FUNCTION_BLOCK FB_IFM_PN2x99
VAR_INPUT
	Grenzwert:REAL; //Grenzwer für HMI Blinken
END_VAR
VAR_OUTPUT
END_VAR
VAR
	IOData AT %I*:INT;
	V12 AT %Q*:BOOL;
	V14 AT %Q*:BOOL;
	
	IOData2:INT;
	Druck:REAL; //mbar (-1000 to 1100)
	OUT1:BOOL;
	OUT2:BOOL;
	
	state:INT:=1;
END_VAR

OUT1:=GETBIT32(inVal32:= IOData, bitNo:= 0);
OUT2:=GETBIT32(inVal32:= IOData, bitNo:= 1);

IOData2:=(IOData/4);
Druck:=INT_TO_REAL(IOData2);
IF Druck>Grenzwert THEN
	MSG_WARNING_List[2]:=TRUE;
END_IF
CASE state OF
	1://off
		V12:=FALSE;
		V14:=FALSE;
	2://wait on
		V12:=TRUE;
		V14:=FALSE;
		state:=3;
	3://on
		V12:=FALSE;
		V14:=FALSE;
	4://wait off
		V12:=FALSE;
		V14:=TRUE;
		state:=1;
	ELSE
		state:=1;
END_CASE

METHOD getPressureString : string
VAR_INPUT
END_VAR
getPressureString:=CONCAT(STR1:=REAL_TO_STRING(Druck), STR2:=' mBar');
END_METHOD

METHOD isActive : BOOL
VAR_INPUT
END_VAR
IF (Druck<Grenzwert) AND state=3 THEN isActive:=TRUE;
ELSIF (Druck>Grenzwert) AND state=3 THEN isActive:=vBlink;
ELSE isActive:=FALSE;
END_IF
END_METHOD

METHOD setState : BOOL
VAR_INPUT
	Enable:BOOL;
END_VAR
IF enable AND state=1 THEN
	state:=2;
ELSIF NOT enable AND state=3 THEN
	state:=4;
END_IF
END_METHOD

END_FUNCTION_BLOCK

(* stored: Version 1.1.0.1, ProductVersion 3.1.4022.9
   POU FB_IFM_PN2x99: Id {9021e297-8ee1-4a86-9c93-5032712ffc9c}, SpecialFunc None
   Method getPressureString: Id {dd23d905-d822-441c-a6e4-424ea0b73e2d}
   Method isActive: Id {4f312e7e-cfa0-4823-ac0b-7b01c37bcf11}
   Method setState: Id {bacb4c47-e79a-4cdd-b97d-37e41eb03924} *)
